(* PLC project Standard Library, Ambitecs Standard Library 1.0, author Lepekhin Igor *)
(* stored: creationDateTime 2024-09-20T00:00:00, modificationDateTime 2024-09-20T08:00:00 *)

TYPE datatype0 : STRUCT
  id : DINT := 1;
  lvl : DINT := 2;
  make : DINT := 3;
END_STRUCT;
END_TYPE

TYPE datatype1 : ARRAY[0..9] OF INT;
END_TYPE

TYPE datatype2 : STRUCT
  one : DINT;
   : ARRAY[0..5] OF WORD;
   : datatype0;
END_STRUCT;
END_TYPE

TYPE datatype3 : BOOL;
END_TYPE

(* The SR bistable is a latch where the Set dominates. *)
FUNCTION_BLOCK SR
  VAR_INPUT
    S1 : BOOL;
    R : BOOL;
  END_VAR
  VAR_OUTPUT
    Q1 : BOOL;
  END_VAR

            Q1 := S1 OR ((NOT R) AND Q1);
          
END_FUNCTION_BLOCK

(* The RS bistable is a latch where the Reset dominates. *)
FUNCTION_BLOCK RS
  VAR_INPUT
    S : BOOL;
    R1 : BOOL;
  END_VAR
  VAR_OUTPUT
    Q1 : BOOL;
  END_VAR

            Q1 := (NOT R1) AND (S OR Q1);
          
END_FUNCTION_BLOCK

(* The semaphore provides a mechanism to allow software elements mutually exclusive access to certain resources. *)
FUNCTION_BLOCK SEMA
  VAR_INPUT
    CLAIM : BOOL;
    RELEASE : BOOL;
  END_VAR
  VAR_OUTPUT
    BUSY : BOOL;
  END_VAR
  VAR
    Q_INTERNAL : BOOL;
  END_VAR

            Q_INTERNAL := CLAIM OR ( Q_INTERNAL AND (NOT RELEASE));
BUSY := Q_INTERNAL;
          
END_FUNCTION_BLOCK

(* The output produces a single pulse when a rising edge is detected. *)
FUNCTION_BLOCK R_TRIG
  VAR_INPUT
    CLK : BOOL;
  END_VAR
  VAR_OUTPUT
    Q : BOOL;
  END_VAR
  VAR RETAIN
    M : BOOL;
  END_VAR

            Q := CLK AND NOT M;
M := CLK;
          
END_FUNCTION_BLOCK

(* The output produces a single pulse when a falling edge is detected. *)
FUNCTION_BLOCK F_TRIG
  VAR_INPUT
    CLK : BOOL;
  END_VAR
  VAR_OUTPUT
    Q : BOOL;
  END_VAR
  VAR RETAIN
    M : BOOL;
  END_VAR

            Q := NOT CLK AND NOT M;
M := NOT CLK;
          
END_FUNCTION_BLOCK

(* The up-counter can be used to signal when a count has reached a maximum value. *)
FUNCTION_BLOCK CTU
  VAR_INPUT
    CU : BOOL;
    R : BOOL;
    PV : INT;
  END_VAR
  VAR_OUTPUT
    Q : BOOL;
    CV : INT;
  END_VAR
  VAR
    CU_T : R_TRIG;
  END_VAR

            CU_T(CU);
IF R THEN CV := 0;
ELSIF CU_T.Q AND (CV < PV)
  THEN CV := CV+1;
END_IF;
Q := (CV >= PV);
          
END_FUNCTION_BLOCK

(* The up-counter can be used to signal when a count has reached a maximum value. *)
FUNCTION_BLOCK CTU_DINT
  VAR_INPUT
    CU : BOOL;
    R : BOOL;
    PV : DINT;
  END_VAR
  VAR_OUTPUT
    Q : BOOL;
    CV : DINT;
  END_VAR
  VAR
    CU_T : R_TRIG;
  END_VAR

            CU_T(CU);
IF R THEN CV := 0;
ELSIF CU_T.Q AND (CV < PV)
  THEN CV := CV+1;
END_IF;
Q := (CV >= PV);
          
END_FUNCTION_BLOCK

(* The up-counter can be used to signal when a count has reached a maximum value. *)
FUNCTION_BLOCK CTU_LINT
  VAR_INPUT
    CU : BOOL;
    R : BOOL;
    PV : LINT;
  END_VAR
  VAR_OUTPUT
    Q : BOOL;
    CV : LINT;
  END_VAR
  VAR
    CU_T : R_TRIG;
  END_VAR

            CU_T(CU);
IF R THEN CV := 0;
ELSIF CU_T.Q AND (CV < PV)
  THEN CV := CV+1;
END_IF;
Q := (CV >= PV);
          
END_FUNCTION_BLOCK

(* The up-counter can be used to signal when a count has reached a maximum value. *)
FUNCTION_BLOCK CTU_UDINT
  VAR_INPUT
    CU : BOOL;
    R : BOOL;
    PV : UDINT;
  END_VAR
  VAR_OUTPUT
    Q : BOOL;
    CV : UDINT;
  END_VAR
  VAR
    CU_T : R_TRIG;
  END_VAR

            CU_T(CU);
IF R THEN CV := 0;
ELSIF CU_T.Q AND (CV < PV)
  THEN CV := CV+1;
END_IF;
Q := (CV >= PV);
          
END_FUNCTION_BLOCK

(* The up-counter can be used to signal when a count has reached a maximum value. *)
FUNCTION_BLOCK CTU_ULINT
  VAR_INPUT
    CU : BOOL;
    R : BOOL;
    PV : ULINT;
  END_VAR
  VAR_OUTPUT
    Q : BOOL;
    CV : ULINT;
  END_VAR
  VAR
    CU_T : R_TRIG;
  END_VAR

            CU_T(CU);
IF R THEN CV := 0;
ELSIF CU_T.Q AND (CV < PV)
  THEN CV := CV+1;
END_IF;
Q := (CV >= PV);
          
END_FUNCTION_BLOCK

(* The down-counter can be used to signal when a count has reached zero, on counting down from a preset value. *)
FUNCTION_BLOCK CTD
  VAR_INPUT
    CD : BOOL;
    LD : BOOL;
    PV : INT;
  END_VAR
  VAR_OUTPUT
    Q : BOOL;
    CV : INT;
  END_VAR
  VAR
    CD_T : R_TRIG;
  END_VAR

            CD_T(CD);
IF LD THEN CV := PV;
ELSIF CD_T.Q AND (CV > 0)
  THEN CV := CV-1;
END_IF;
Q := (CV <= 0);
          
END_FUNCTION_BLOCK

(* The down-counter can be used to signal when a count has reached zero, on counting down from a preset value. *)
FUNCTION_BLOCK CTD_DINT
  VAR_INPUT
    CD : BOOL;
    LD : BOOL;
    PV : DINT;
  END_VAR
  VAR_OUTPUT
    Q : BOOL;
    CV : DINT;
  END_VAR
  VAR
    CD_T : R_TRIG;
  END_VAR

            CD_T(CD);
IF LD THEN CV := PV;
ELSIF CD_T.Q AND (CV > 0)
  THEN CV := CV-1;
END_IF;
Q := (CV <= 0);
          
END_FUNCTION_BLOCK

(* The down-counter can be used to signal when a count has reached zero, on counting down from a preset value. *)
FUNCTION_BLOCK CTD_LINT
  VAR_INPUT
    CD : BOOL;
    LD : BOOL;
    PV : LINT;
  END_VAR
  VAR_OUTPUT
    Q : BOOL;
    CV : LINT;
  END_VAR
  VAR
    CD_T : R_TRIG;
  END_VAR

            CD_T(CD);
IF LD THEN CV := PV;
ELSIF CD_T.Q AND (CV > 0)
  THEN CV := CV-1;
END_IF;
Q := (CV <= 0);
          
END_FUNCTION_BLOCK

(* The down-counter can be used to signal when a count has reached zero, on counting down from a preset value. *)
FUNCTION_BLOCK CTD_UDINT
  VAR_INPUT
    CD : BOOL;
    LD : BOOL;
    PV : UDINT;
  END_VAR
  VAR_OUTPUT
    Q : BOOL;
    CV : UDINT;
  END_VAR
  VAR
    CD_T : R_TRIG;
  END_VAR

            CD_T(CD);
IF LD THEN CV := PV;
ELSIF CD_T.Q AND (CV > 0)
  THEN CV := CV-1;
END_IF;
Q := (CV <= 0);
          
END_FUNCTION_BLOCK

(* The down-counter can be used to signal when a count has reached zero, on counting down from a preset value. *)
FUNCTION_BLOCK CTD_ULINT
  VAR_INPUT
    CD : BOOL;
    LD : BOOL;
    PV : ULINT;
  END_VAR
  VAR_OUTPUT
    Q : BOOL;
    CV : ULINT;
  END_VAR
  VAR
    CD_T : R_TRIG;
  END_VAR

            CD_T(CD);
IF LD THEN CV := PV;
ELSIF CD_T.Q AND (CV > 0)
  THEN CV := CV-1;
END_IF;
Q := (CV <= 0);
          
END_FUNCTION_BLOCK

(* The up-down counter has two inputs CU and CD. It can be used to both count up on one input and down on the other. *)
FUNCTION_BLOCK CTUD
  VAR_INPUT
    CU : BOOL;
    CD : BOOL;
    R : BOOL;
    LD : BOOL;
    PV : INT;
  END_VAR
  VAR_OUTPUT
    QU : BOOL;
    QD : BOOL;
    CV : INT;
    CD_T : R_TRIG;
    CU_T : R_TRIG;
  END_VAR

            CD_T(CD);
CU_T(CU);
IF R THEN CV := 0;
ELSIF LD THEN CV := PV;
ELSE
  IF NOT (CU_T.Q AND CD_T.Q) THEN
    IF CU_T.Q AND (CV < PV)
    THEN CV := CV+1;
    ELSIF CD_T.Q AND (CV > 0)
    THEN CV := CV-1;
    END_IF;
  END_IF;
END_IF;
QU := (CV >= PV);
QD := (CV <= 0);
          
END_FUNCTION_BLOCK

(* The up-down counter has two inputs CU and CD. It can be used to both count up on one input and down on the other. *)
FUNCTION_BLOCK CTUD_DINT
  VAR_INPUT
    CU : BOOL;
    CD : BOOL;
    R : BOOL;
    LD : BOOL;
    PV : DINT;
  END_VAR
  VAR_OUTPUT
    QU : BOOL;
    QD : BOOL;
    CV : DINT;
    CD_T : R_TRIG;
    CU_T : R_TRIG;
  END_VAR

            CD_T(CD);
CU_T(CU);
IF R THEN CV := 0;
ELSIF LD THEN CV := PV;
ELSE
  IF NOT (CU_T.Q AND CD_T.Q) THEN
    IF CU_T.Q AND (CV < PV)
    THEN CV := CV+1;
    ELSIF CD_T.Q AND (CV > 0)
    THEN CV := CV-1;
    END_IF;
  END_IF;
END_IF;
QU := (CV >= PV);
QD := (CV <= 0);
          
END_FUNCTION_BLOCK

(* The up-down counter has two inputs CU and CD. It can be used to both count up on one input and down on the other. *)
FUNCTION_BLOCK CTUD_LINT
  VAR_INPUT
    CU : BOOL;
    CD : BOOL;
    R : BOOL;
    LD : BOOL;
    PV : LINT;
  END_VAR
  VAR_OUTPUT
    QU : BOOL;
    QD : BOOL;
    CV : LINT;
    CD_T : R_TRIG;
    CU_T : R_TRIG;
  END_VAR

            CD_T(CD);
CU_T(CU);
IF R THEN CV := 0;
ELSIF LD THEN CV := PV;
ELSE
  IF NOT (CU_T.Q AND CD_T.Q) THEN
    IF CU_T.Q AND (CV < PV)
    THEN CV := CV+1;
    ELSIF CD_T.Q AND (CV > 0)
    THEN CV := CV-1;
    END_IF;
  END_IF;
END_IF;
QU := (CV >= PV);
QD := (CV <= 0);
          
END_FUNCTION_BLOCK

(* The up-down counter has two inputs CU and CD. It can be used to both count up on one input and down on the other. *)
FUNCTION_BLOCK CTUD_UDINT
  VAR_INPUT
    CU : BOOL;
    CD : BOOL;
    R : BOOL;
    LD : BOOL;
    PV : UDINT;
  END_VAR
  VAR_OUTPUT
    QU : BOOL;
    QD : BOOL;
    CV : UDINT;
    CD_T : R_TRIG;
    CU_T : R_TRIG;
  END_VAR

            CD_T(CD);
CU_T(CU);
IF R THEN CV := 0;
ELSIF LD THEN CV := PV;
ELSE
  IF NOT (CU_T.Q AND CD_T.Q) THEN
    IF CU_T.Q AND (CV < PV)
    THEN CV := CV+1;
    ELSIF CD_T.Q AND (CV > 0)
    THEN CV := CV-1;
    END_IF;
  END_IF;
END_IF;
QU := (CV >= PV);
QD := (CV <= 0);
          
END_FUNCTION_BLOCK

(* The up-down counter has two inputs CU and CD. It can be used to both count up on one input and down on the other. *)
FUNCTION_BLOCK CTUD_ULINT
  VAR_INPUT
    CU : BOOL;
    CD : BOOL;
    R : BOOL;
    LD : BOOL;
    PV : ULINT;
  END_VAR
  VAR_OUTPUT
    QU : BOOL;
    QD : BOOL;
    CV : ULINT;
    CD_T : R_TRIG;
    CU_T : R_TRIG;
  END_VAR

            CD_T(CD);
CU_T(CU);
IF R THEN CV := 0;
ELSIF LD THEN CV := PV;
ELSE
  IF NOT (CU_T.Q AND CD_T.Q) THEN
    IF CU_T.Q AND (CV < PV)
    THEN CV := CV+1;
    ELSIF CD_T.Q AND (CV > 0)
    THEN CV := CV-1;
    END_IF;
  END_IF;
END_IF;
QU := (CV >= PV);
QD := (CV <= 0);
          
END_FUNCTION_BLOCK

(* The pulse timer can be used to generate output pulses of a given time duration. *)
FUNCTION_BLOCK TP
  VAR_INPUT
    IN : BOOL;  (* first input parameter *)
    PT : TIME;  (* second input parameter *)
  END_VAR
  VAR_OUTPUT
    Q : BOOL := FALSE;  (* first output parameter *)
    ET : TIME := T#0s;  (* second output parameter *)
  END_VAR
  VAR
    STATE : SINT := 0;  (* internal state: 0-reset, 1-counting, 2-set *)
    PREV_IN : BOOL := FALSE;
    CURRENT_TIME : TIME;
    START_TIME : TIME;
  END_VAR

            {__SET_VAR(data__->,CURRENT_TIME,,__CURRENT_TIME)}

IF ((STATE = 0) AND NOT(PREV_IN) AND IN)   (* found rising edge on IN *)
THEN
  (* start timer... *)
  STATE := 1;
  Q := TRUE;
  START_TIME := CURRENT_TIME;

ELSIF (STATE = 1)
THEN
  IF ((START_TIME + PT) <= CURRENT_TIME)
  THEN
    STATE := 2;
    Q := FALSE;
    ET := PT;
  ELSE
    ET := CURRENT_TIME - START_TIME;
  END_IF;
END_IF;

IF ((STATE = 2) AND NOT(IN))
THEN
  ET := T#0s;
  STATE := 0;
END_IF;

PREV_IN := IN;

          
END_FUNCTION_BLOCK

(* The on-delay timer can be used to delay setting an output true, for fixed period after an input becomes true. *)
FUNCTION_BLOCK TON
  VAR_INPUT
    IN : BOOL;  (* first input parameter *)
    PT : TIME;  (* second input parameter *)
  END_VAR
  VAR_OUTPUT
    Q : BOOL := FALSE;  (* first output parameter *)
    ET : TIME := T#0s;  (* second output parameter *)
  END_VAR
  VAR
    STATE : SINT := 0;  (* internal state: 0-reset, 1-counting, 2-set *)
    PREV_IN : BOOL := FALSE;
    CURRENT_TIME : TIME;
    START_TIME : TIME;
  END_VAR

            {__SET_VAR(data__->,CURRENT_TIME,,__CURRENT_TIME)}

IF ((STATE = 0) AND NOT(PREV_IN) AND IN)   (* found rising edge on IN *)
THEN
  (* start timer... *)
  STATE := 1;
  Q := FALSE;
  START_TIME := CURRENT_TIME;

ELSE
  (* STATE is 1 or 2 !! *)
  IF (NOT(IN))
  THEN
    ET := T#0s;
    Q := FALSE;
    STATE := 0;

  ELSIF (STATE = 1)
  THEN
    IF ((START_TIME + PT) <= CURRENT_TIME)
    THEN
      STATE := 2;
      Q := TRUE;
      ET := PT;
    ELSE
      ET := CURRENT_TIME - START_TIME;
    END_IF;
  END_IF;

END_IF;

PREV_IN := IN;

          
END_FUNCTION_BLOCK

(* The off-delay timer can be used to delay setting an output false, for fixed period after input goes false. *)
FUNCTION_BLOCK TOF
  VAR_INPUT
    IN : BOOL;  (* first input parameter *)
    PT : TIME;  (* second input parameter *)
  END_VAR
  VAR_OUTPUT
    Q : BOOL := FALSE;  (* first output parameter *)
    ET : TIME := T#0s;  (* second output parameter *)
  END_VAR
  VAR
    STATE : SINT := 0;  (* internal state: 0-reset, 1-counting, 2-set *)
    PREV_IN : BOOL := FALSE;
    CURRENT_TIME : TIME;
    START_TIME : TIME;
  END_VAR

            {__SET_VAR(data__->,CURRENT_TIME,,__CURRENT_TIME)}

IF ((STATE = 0) AND PREV_IN AND NOT(IN))   (* found falling edge on IN *)
THEN
  (* start timer... *)
  STATE := 1;
  START_TIME := CURRENT_TIME;

ELSE
  (* STATE is 1 or 2 !! *)
  IF (IN)
  THEN
    ET := T#0s;
    STATE := 0;

  ELSIF (STATE = 1)
  THEN
    IF ((START_TIME + PT) <= CURRENT_TIME)
    THEN
      STATE := 2;
      ET := PT;
    ELSE
      ET := CURRENT_TIME - START_TIME;
    END_IF;
  END_IF;

END_IF;

Q := IN OR (STATE = 1);
PREV_IN := IN;

          
END_FUNCTION_BLOCK
